Fanuc KAREL source: ka00014.KL

-- PROVISIONAL review KL for V770-1; original PC SHA256 2c4cbc3b2805759f281d983d5bd9ae48c2dd53cb453db9fe1dac8edbe9a142a6
-- Incomplete behavior may be omitted. Consult companion uncertainty JSON. Do not deploy.
PROGRAM KA00014
%NOLOCKGROUP
VAR
  SRC : REAL
  DST : REAL
BEGIN
  -- UNRESOLVED_PC offsets 5-16; opcodes 2E,23
  -- UNRESOLVED_PC offsets 21-33; opcodes 21,23
  -- UNRESOLVED_PC offsets 38-42; opcodes 7F
END KA00014
